// TIA Portal V19 export
TYPE "PPrf_CoilHandling_WeldingCycle"
// stored: Access Published
   STRUCT
      MeasureSheetEdgeReference : LReal;   // Distance of sheet edge from reference
      CorrStartWelding : LReal;   // Start welding correction absolute value
      CorrStopWelding : LReal;   // Stop welding correction absolute value
   END_STRUCT;
END_TYPE
